Fanuc KAREL source: SET_LANG.kl

PROGRAM T
%NOLOCKGROUP
VAR
 v0 : STRING[40]
 v1 : INTEGER
BEGIN
 SET_LANG(v0, v1)
END T
